{attribute 'qualified_only'}
{attribute 'strict'}
TYPE E_CarrierType :
(
	EM4102		:= 16#3032,
	EM4550		:= 16#3033,
	Nova		:= 16#3130,
	Q5			:= 16#3131,
	T5557		:= 16#3134,
	MDT_28		:= 16#3135,
	ISO15693	:= 16#3230,
	MDT_112		:= 16#3231,
	TiHF_I		:= 16#3232,
	SRF55V02P	:= 16#3233,
	SRF55V10P	:= 16#3234,
	MDT_2K_H	:= 16#3333,
	SLI_S		:= 16#3335,
	Depending	:= 16#3939
)WORD := MDT_28;
END_TYPE
//  EM4102 = '16#3032'
//  EM4550 = '16#3033'
//  Nova = '16#3130'
//  Q5 = '16#3131'
//  T5557 = '16#3134'
//  MDT_28 = '16#3135'
//  ISO15693 = '16#3230'
//  MDT_112 = '16#3231'
//  TiHF_I = '16#3232'
//  SRF55V02P = '16#3233'
//  SRF55V10P = '16#3234'
//  MDT_2K_H = '16#3333'
//  SLI_S = '16#3335'
//  Depending = '16#3939'

(* stored: Version 1.1.0.1, ProductVersion 3.1.4024.11
   EnumerationTextList E_CarrierType: Id {0efa1e39-f5cb-42f4-97d9-78560f31c819} *)
